PROGRAM MAIN
VAR
	Station : Wrapper;
	
	ActInputs	: ActInputs;
	ActOutputs	: ActOutputs;
	Buttons		: Buttons;
	Flags		: Flags;
END_VAR

Station(ActInputs 	:= ActInputs,
		ActOutputs	=> ActOutputs,
		Buttons		:= Buttons,
		Flags		=> Flags);

END_PROGRAM

(* stored: Version 1.1.0.1, ProductVersion 3.1.4024.9
   POU MAIN: Id {259cb9c3-c65a-4752-87a5-cbb355eff08d}, SpecialFunc None *)
